(* CoDeSys 2.3.9.41 project: wwww.pro *)
(* Libraries: STANDARD.LIB 4.10.05 11:14:46, IECSFC.LIB 13.4.06 15:51:28, SYSLIBTIME.LIB 20.2.06 13:31:16, SYSTASKINFO.LIB 20.2.06 13:31:38, ANALYZATION.LIB 5.10.99 09:05:06, SYSLIBCALLBACK.LIB 20.2.06 13:31:08 *)

(* PLC configuration (modules and I/O channels)
PLC110_32 [Root] node -1, in %IB0 out %QB0 {MinCycleLength = 1; MaxCycleLength = 1000; MaxBackupTime = 6}
  Fast discrete inputs [I_SIMPLE_INPUT] node 0, in %IB0 out %QB0 {Filtrationtime = 10; Visibility = No}
    AT %IX0.0 [BitInput] Discrete input 1
    AT %IX0.1 [BitInput] Discrete input 2
x AT %IB1.0 [ByteInput] 8 discrete inputs
z AT %IB1.1 [ByteInput] 8 discrete inputs
Fast discrete outputs [OWEN_ID570] node 2, in %IB2 out %QB2 {SafeValueBool = FALSE; SafeValueBool = FALSE; SafeValueBool = FALSE; SafeValueBool = FALSE; Visibility = No}
  AT %QX2.0 [BitOutput] Fast discrete output 1
  AT %QX2.1 [BitOutput] Fast discrete output 2
  AT %QX2.2 [BitOutput] Fast discrete output 3
  AT %QX2.3 [BitOutput] Fast discrete output 4
y AT %QB3.0 [ByteOutput] 8 discrete outputs
q AT %QB3.1 [ByteOutput] 2 discrete outputs
Special input [ID103] node 4, in %IB4 out %QB4 {Filtrationtime = 1000; PinCount = 1; WatchDogPeriod = 400; PollPeriod = 3000; Visibility = No}
  AT %IX4.0 [BitInput] Special input
Special output [ID104] node 5, in %IB5 out %QB5 {Visibility = No; PinCount = 1}
  AT %QX5.0 [BitOutput] Special output
TCP [TCP_ID221] node 0, in %IB6.0.0 out %QB6.0.0 {RemotePort = 502; Visibility = No}
v AT %QB6.1.0 [ByteOutput]
w AT %QB6.2.0 [ByteOutput]
c AT %QW6.3.0 [WordOutput]
d AT %QW6.4.0 [WordOutput]
*)

(* POU PLC_PRG, LD *)
PROGRAM PLC_PRG
VAR
	N: TIME;
	www: TIME;
	uuuu: TON;
	qqq: TOF;
	g: TIME;
	eeee: TOF;
	wwww: TOF;
	k: TIME;
END_VAR
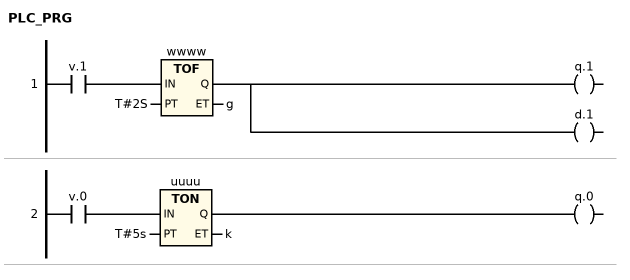
_LD_ (* Ladder Diagram *)
NETWORK 1
	[v.1] - wwww:TOF(IN: *, PT: T#2S, ET => g) --- (q.1) (d.1)
NETWORK 2
	[v.0] - uuuu:TON(IN: *, PT: T#5s, ET => k) --- (q.0)
_END_LD_
(* the same logic as Structured Text *)
(* Network 1 *)
wwww(IN := v.1, PT := T#2S);
g := wwww.ET;
q.1 := wwww.Q;
d.1 := wwww.Q;
(* Network 2 *)
uuuu(IN := v.0, PT := T#5s);
k := uuuu.ET;
q.0 := uuuu.Q;
END_PROGRAM
